// TwinCAT 3 PLC project _1_00
// ProgramVersion: 3.1.4023.0
// libraries:
//   Tc2_Standard, * (Beckhoff Automation GmbH)
//   Tc2_System, * (Beckhoff Automation GmbH)
//   Tc3_Module, * (Beckhoff Automation GmbH)
// project tree:
//   01_SubModule/01_Unit/ E_Unit.TcDUT, ST_Unit.TcDUT
//   01_SubModule/02_Station/ FB_Station.TcPOU
//   02_Module/ FB_Arm.TcPOU, FB_Barn.TcPOU, FB_Breeder.TcPOU, FB_Incubator.TcPOU, FB_Market.TcPOU
//   03_Game/ FB_Game.TcPOU
//   04_Main/ MAIN.TcPOU
//   / PlcTask.TcTTO
// real-time tasks:
//   TASK PlcTask: cycle T#10ms, priority 20, ADS port 350

CONFIGURATION _1_00
    RESOURCE PLC ON TwinCAT3
        TASK PlcTask(INTERVAL := T#10ms, PRIORITY := 20);
        PROGRAM MAIN WITH PlcTask : MAIN;
    END_RESOURCE
END_CONFIGURATION

// ---- 01_SubModule/01_Unit/E_Unit.TcDUT
{attribute 'qualified_only'}
{attribute 'strict'}
TYPE E_Unit :
(
	Invalid := -1,
	Egg		:= 0,
	Chicken	:= 1
):= Invalid;
END_TYPE

// ---- 01_SubModule/01_Unit/ST_Unit.TcDUT
TYPE ST_Unit :
STRUCT
	eType		: E_Unit;
	iHitPoint	: INT;
	iProgress	: INT;
END_STRUCT
END_TYPE

// ---- 04_Main/MAIN.TcPOU
PROGRAM MAIN
VAR
	(**)
	fbGame			: FB_Game;
	(*Button*)
	btStart			: BOOL;
	btPause			: BOOL;
	(*State*)
	GameRunning			: BOOL;
END_VAR

IF btStart THEN
	btStart := NOT btStart;
	GameRunning := TRUE;
END_IF

IF btPause THEN
	btPause := NOT btPause;
	GameRunning := FALSE;
END_IF

IF GameRunning THEN
	fbGame();
END_IF

END_PROGRAM

// ---- 03_Game/FB_Game.TcPOU
FUNCTION_BLOCK FB_Game
VAR
(*===========================================================================================================================*)
	(*Buttons*)
		(*Transfer*)
	btBarnToBreeder			: BOOL;
	btBarnToIncubator		: BOOL;
	btSellEgg				: BOOL;
	btSellChicken			: BOOL;
	btBreederToBarn			: BOOL;
	btPurchaseEgg			: BOOL;
	btPurchaseChicken		: BOOL;
		(*Upgrades*)
	btUpgradeArm			: BOOL;
	btUpgradeBarn			: BOOL;
	btUpgradeBreeder		: BOOL;
	btUpgradeIncubator		: BOOL;
	btUpgradeMarket			: BOOL;
	(*/Buttons*)
(*===========================================================================================================================*)
	(*Instance*)
		(*Stations*)
	fbBarn					: FB_Barn;
	fbBreeder				: FB_Breeder;
	fbIncubator				: FB_Incubator;
	fbMarket				: FB_Market;
		(*Arms*)
	fbArmArr				: ARRAY [1..5] OF FB_Arm;
	iCurArmLevel			: INT;
	iMaxArmLevel			: INT;
		(*Status*)
	iDay					: INT;
	iHour					: INT;
	iCurrency				: INT;
	iCost					: INT;
	iBarnUnit				: INT;
	iBreederUnit			: INT;
	iIncubatorUnit			: INT;
	iMarketUnit				: INT;
		(*Game Setting*)
	MaxStationLevel			: INT	:= 5;
	BarnLocation			: REAL	:= 10;
	BreederLocation			: REAL	:= 50;
	IncubatorLocation		: REAL	:= 90;
	MarketLocation			: REAL	:= 130;
	InitArmX				: REAL	:= 0;
	InitArmY				: REAL	:= 0;
	
		(*Timer*)
	fbTon60FPS				: TON;
	fbTon30FPS				: TON;
	fbTon1S					: TON;
	(*/Instance*)
END_VAR

Initialize(MaxStationLevel, BarnLocation, BreederLocation, IncubatorLocation, MarketLocation, 100);

fbTon30FPS(IN:= TRUE, PT:= T#33MS);
IF fbTon30FPS.Q THEN
	fbTon30FPS(IN:= FALSE);
	
	fbBarn.SortDescending();
	fbBreeder.SortAscending();
	fbIncubator.SortAscending();
	
	ButtonsTransfer();
	ArmRun();
	
	iBarnUnit := fbBarn.TotalUnit;
	iBreederUnit := fbBreeder.TotalUnit;
	iIncubatorUnit := fbIncubator.TotalUnit;
	iMarketUnit := fbMarket.TotalUnit;
	
END_IF

fbTon1S(IN:= TRUE, PT:= T#1S);
IF fbTon1S.Q THEN
	fbTon1S(IN:= FALSE);
	
	fbBarn.Run();
	fbBarn.HpRecover();
	
	fbBreeder.Run();
	fbBreeder.HpDeduct();
	
	fbIncubator.Run();
	
	fbMarket.Run();
	
	fbBarn.AutoImport(fbBreeder.Breeding(), fbIncubator.Hatching());
	iCurrency := iCurrency + fbMarket.Marketing();
	
	iHour := iHour + 1;
END_IF

IF iHour > 23 THEN
	iHour := 0;
	iDay := iDay + 1;
	iCurrency := iCurrency - iCost;
	IF iCurrency >= 0 THEN
		iCost := iCost + iDay*10;
	ELSE
		// Lose
	END_IF
	
END_IF

IF iDay > 30 THEN
	// Win
END_IF

METHOD ArmRun : PVOID
VAR
	iIndex			: INT;
END_VAR
fbArmArr[1].Run();
fbArmArr[2].Run();
fbArmArr[3].Run();
fbArmArr[4].Run();
fbArmArr[5].Run();

FOR iIndex := 1 TO iCurArmLevel BY 1 DO
	IF fbArmArr[iIndex].Load THEN
		IF
			fbArmArr[iIndex].CurX = fbBarn.Location THEN
			IF
				fbArmArr[iIndex].UnitType = 0 THEN
				fbArmArr[iIndex].CurUnit := fbBarn.UnitExport(0);
				fbArmArr[iIndex].Load := FALSE;
			ELSIF
				fbArmArr[iIndex].UnitType = 1 THEN
				fbArmArr[iIndex].CurUnit := fbBarn.UnitExport(1);
				fbArmArr[iIndex].Load := FALSE;
			END_IF
		ELSIF
			fbArmArr[iIndex].CurX = fbBreeder.Location THEN
			IF
				fbArmArr[iIndex].UnitType = 1 THEN
				fbArmArr[iIndex].CurUnit := fbBreeder.UnitExport(1);
				fbArmArr[iIndex].Load := FALSE;
			END_IF
		END_IF
	END_IF
END_FOR

FOR iIndex := 1 TO iCurArmLevel BY 1 DO
	IF fbArmArr[iIndex].Unload THEN
		IF
			fbArmArr[iIndex].CurX = fbBarn.Location THEN
			fbBarn.UnitImport(fbArmArr[iIndex].CurUnit);
			fbArmArr[iIndex].Unload := FALSE;
		ELSIF
			fbArmArr[iIndex].CurX = fbBreeder.Location THEN
			fbBreeder.UnitImport(fbArmArr[iIndex].CurUnit);
			fbArmArr[iIndex].Unload := FALSE;
		ELSIF
			fbArmArr[iIndex].CurX = fbIncubator.Location THEN
			fbIncubator.UnitImport(fbArmArr[iIndex].CurUnit);
			fbArmArr[iIndex].Unload := FALSE;
		ELSIF
			fbArmArr[iIndex].CurX = fbMarket.Location THEN
			fbMarket.UnitImport(fbArmArr[iIndex].CurUnit);
			fbArmArr[iIndex].Unload := FALSE;
		END_IF
	END_IF
END_FOR
END_METHOD

METHOD ButtonsTransfer : PVOID
VAR
	stTempUnit			: ST_Unit;
END_VAR
IF btBarnToBreeder THEN
	btBarnToBreeder := NOT btBarnToBreeder;
	
	IF NOT fbBreeder.IsFull AND fbBarn.HasChicken THEN
		TransferUnit(fbBarn.Location, fbBreeder.Location, 1);
	END_IF
END_IF

IF btBarnToIncubator THEN
	btBarnToIncubator := NOT btBarnToIncubator;
	
	IF NOT fbIncubator.IsFull AND fbBarn.HasEgg  THEN
		TransferUnit(fbBarn.Location, fbIncubator.Location, 0);
	END_IF
END_IF

IF btSellEgg THEN
	btSellEgg := NOT btSellEgg;
	
	IF NOT fbMarket.IsFull AND fbBarn.HasEgg THEN
		TransferUnit(fbBarn.Location, fbMarket.Location, 0);
	END_IF	
END_IF

IF btSellChicken THEN
	btSellChicken := NOT btSellChicken;
	
	IF NOT fbMarket.IsFull AND fbBarn.HasChicken THEN
		TransferUnit(fbBarn.Location, fbMarket.Location, 1);
	END_IF	
END_IF

IF btBreederToBarn THEN
	btBreederToBarn := NOT btBreederToBarn;
	
	IF NOT fbBarn.IsFull AND fbBreeder.HasChicken THEN
		TransferUnit(fbBreeder.Location, fbBarn.Location, 1);
	END_IF
END_IF

IF btPurchaseEgg THEN
	btPurchaseEgg := NOT btPurchaseEgg;
	
	IF NOT fbBarn.IsFull AND iCurrency > 20 THEN
		iCurrency := iCurrency - 20;
		
		stTempUnit.eType := 0;
		stTempUnit.iHitPoint := 30;
		stTempUnit.iProgress := 0;
		fbBarn.UnitImport(stTempUnit);
	END_IF
END_IF

IF btPurchaseChicken THEN
	btPurchaseChicken := NOT btPurchaseChicken;
	
	IF  NOT fbBarn.IsFull AND iCurrency > 12 THEN
		iCurrency := iCurrency - 12;
		
		stTempUnit.eType := 1;
		stTempUnit.iHitPoint := 30;
		stTempUnit.iProgress := 0;
		fbBarn.UnitImport(stTempUnit);
	END_IF
END_IF
END_METHOD

METHOD ButtonsUpgrade : PVOID
VAR_INPUT
END_VAR
IF btUpgradeArm THEN
	btUpgradeArm := NOT btUpgradeArm;
	
	IF iCurrency > (iCurArmLevel*30) THEN
		iCurrency := iCurrency - (iCurArmLevel*30);
		UpgradeArm(iCurArmLevel, InitArmX, InitArmY);
	END_IF
END_IF

IF btUpgradeBarn THEN
	btUpgradeBarn := NOT btUpgradeBarn;
	
	IF iCurrency > (fbBarn.Level*30) THEN
		iCurrency := iCurrency - (fbBarn.Level*30);
		fbBarn.Upgrade();
	END_IF
END_IF

IF btUpgradeBreeder THEN
	btUpgradeBreeder := NOT btUpgradeBreeder;
	
	IF iCurrency > (fbBreeder.Level*30) THEN
		iCurrency := iCurrency - (fbBreeder.Level*30);
		fbBreeder.Upgrade();
	END_IF
END_IF

IF btUpgradeIncubator THEN
	btUpgradeIncubator := NOT btUpgradeIncubator;
	
	IF iCurrency > (fbIncubator.Level*30) THEN
		iCurrency := iCurrency - (fbIncubator.Level*30);
		fbIncubator.Upgrade();
	END_IF
END_IF

IF btUpgradeMarket THEN
	btUpgradeMarket := NOT btUpgradeMarket;
	
	IF iCurrency > (fbMarket.Level*30) THEN
		iCurrency := iCurrency - (fbMarket.Level*30);
		fbMarket.Upgrade();
	END_IF
END_IF
END_METHOD

METHOD Initialize : PVOID
VAR_INPUT
	MaxLevel					: INT;
	BarnLocation				: REAL;
	BreederLocation				: REAL;
	IncubatorLocation			: REAL;
	MarketLocation				: REAL;
	Currency					: INT;
END_VAR
IF iDay = 0 THEN
	iDay := 1;
	
	fbBarn.Set(MaxLevel, BarnLocation);
	fbBreeder.Set(MaxLevel, BreederLocation);
	fbIncubator.Set(MaxLevel, IncubatorLocation);
	fbMarket.Set(MaxLevel, MarketLocation);
	UpgradeArm(iCurArmLevel, InitArmX, InitArmY);
	
	iCurrency := Currency;
	iCost := 10;
END_IF
END_METHOD

METHOD TransferUnit : PVOID
VAR_INPUT
	ImportLocation			: REAL;
	ExportLocation			: REAL;
	UnitType				: INT;	//0: Egg, 1: Chicken
END_VAR
VAR
	iIndex					: INT;
END_VAR
FOR iIndex := 1 TO iCurArmLevel BY 1 DO
	IF fbArmArr[iIndex].Activated AND NOT fbArmArr[iIndex].Busy THEN
		fbArmArr[iIndex].Assign(ImportLocation, ExportLocation, UnitType);
		RETURN;
	END_IF
END_FOR
END_METHOD

METHOD UpgradeArm : PVOID
VAR_INPUT
	CurrentArmIndex		: INT;
	InitX				: REAL;
	InitY				: REAL;
END_VAR
CurrentArmIndex := CurrentArmIndex + 1;
fbArmArr[CurrentArmIndex].Activated := TRUE;
fbArmArr[CurrentArmIndex].CurX := InitX;
fbArmArr[CurrentArmIndex].CurX := InitY;
iCurArmLevel := CurrentArmIndex;
END_METHOD

END_FUNCTION_BLOCK

// ---- 02_Module/FB_Barn.TcPOU
FUNCTION_BLOCK FB_Barn EXTENDS FB_Station
VAR
END_VAR

METHOD AutoImport : PVOID
VAR_INPUT
	Egg			: INT;
	Chicken		: INT;
END_VAR
VAR
	stTempEgg			: ST_Unit;
	iTempEgg			: INT;
	stTempChicken		: ST_Unit;
	iTempChicken		: INT;
END_VAR
FOR iTempEgg := 1 TO Egg BY 1 DO
	stTempEgg.eType := 0;
	stTempEgg.iHitPoint := 30;
	stTempEgg.iProgress := 0;
	UnitImport(stTempEgg);
END_FOR

FOR iTempChicken := 1 TO Chicken BY 1 DO
	stTempChicken.eType := 1;
	stTempChicken.iHitPoint := 30;
	stTempChicken.iProgress := 0;
	UnitImport(stTempChicken);
END_FOR
END_METHOD

METHOD Run : BOOL
VAR_INPUT
END_VAR
iMaxUnit := iCurLevel * 20;
END_METHOD

END_FUNCTION_BLOCK

// ---- 01_SubModule/02_Station/FB_Station.TcPOU
FUNCTION_BLOCK FB_Station
VAR
	stUnitArr			: ARRAY [1..100] OF ST_Unit;
	iMaxUnit			: INT;
	iLastIndex			: INT;
	
	iMaxLevel			: INT;
	iCurLevel			: INT := 1;
	
	rLocation			: REAL;
END_VAR

PROPERTY HasChicken : BOOL
GET
VAR
	iIndex			: INT;
END_VAR
HasChicken := FALSE;
IF iLastIndex > 0 THEN
	FOR iIndex := 1 TO iLastIndex BY 1 DO
		IF stUnitArr[iIndex].eType = 1 THEN
			HasChicken := NOT HasChicken;
			RETURN;
		END_IF
	END_FOR
END_IF
END_GET
END_PROPERTY

PROPERTY HasEgg : BOOL
GET
VAR
	iIndex			: INT;
END_VAR
HasEgg := FALSE;
IF iLastIndex > 0 THEN
	FOR iIndex := 1 TO iLastIndex BY 1 DO
		IF stUnitArr[iIndex].eType = 0 THEN
			HasEgg := NOT HasEgg;
			RETURN;
		END_IF
	END_FOR
END_IF
END_GET
END_PROPERTY

METHOD HpDeduct : PVOID
VAR
	iTempIndex			: INT;
END_VAR
IF iLastIndex < 1 THEN
	RETURN;
END_IF

FOR iTempIndex := 1 TO iLastIndex BY 1 DO
	stUnitArr[iTempIndex].iHitPoint := stUnitArr[iTempIndex].iHitPoint - 1;
	IF stUnitArr[iTempIndex].iHitPoint = 0 THEN
		RemoveUnit(iTempIndex);
	END_IF
END_FOR
END_METHOD

METHOD HpRecover : PVOID
VAR
	iTempIndex			: INT;
END_VAR
IF iLastIndex < 1 THEN
	RETURN;
END_IF

FOR iTempIndex := 1 TO iLastIndex BY 1 DO
	IF stUnitArr[iTempIndex].iHitPoint < 30 THEN
		stUnitArr[iTempIndex].iHitPoint := stUnitArr[iTempIndex].iHitPoint + 1;
	END_IF
END_FOR
END_METHOD

PROPERTY IsFull : BOOL
GET
IsFull := TRUE;
IF iLastIndex < iMaxUnit THEN
	IsFull := NOT IsFull;
END_IF
END_GET
END_PROPERTY

PROPERTY Level : INT
GET
Level := iCurLevel;
END_GET
END_PROPERTY

PROPERTY Location : REAL
GET
Location := rLocation;
END_GET
END_PROPERTY

METHOD RemoveUnit : PVOID
VAR_INPUT
	iIndex			: INT;
END_VAR
stUnitArr[iIndex] := stUnitArr[iLastIndex];
stUnitArr[iLastIndex].eType := -1;
stUnitArr[iLastIndex].iHitPoint := 0;
stUnitArr[iLastIndex].iProgress := 0;
iLastIndex := iLastIndex - 1;
END_METHOD

METHOD Run : BOOL
VAR_INPUT
END_VAR
iMaxUnit := iCurLevel * 10;
END_METHOD

METHOD Set : PVOID
VAR_INPUT
	MaxLevel			: INT;
	Location			: REAL;
END_VAR
iMaxLevel := MaxLevel;
rLocation := Location;
iCurLevel := 1;
END_METHOD

METHOD SortAscending : PVOID
VAR
	iCurIndex			: INT;
	stTempUnit			: ST_Unit;
	iTempIndex			: INT;
END_VAR
IF iLastIndex < 2 THEN
	RETURN;
END_IF

FOR iTempIndex := 1 TO iLastIndex BY 1 DO
	FOR iCurIndex := 1 TO iLastIndex BY 1 DO
		IF stUnitArr[iCurIndex].iHitPoint > stUnitArr[iTempIndex].iHitPoint THEN
			stTempUnit := stUnitArr[iCurIndex];
			stUnitArr[iCurIndex] := stUnitArr[iTempIndex];
			stUnitArr[iTempIndex] := stTempUnit;
		END_IF
	END_FOR
END_FOR
END_METHOD

METHOD SortDescending : PVOID
VAR
	iCurIndex			: INT;
	stTempUnit			: ST_Unit;
	iTempIndex			: INT;
END_VAR
IF iLastIndex < 2 THEN
	RETURN;
END_IF

FOR iTempIndex := 1 TO iLastIndex BY 1 DO
	FOR iCurIndex := 1 TO iLastIndex BY 1 DO
		IF stUnitArr[iCurIndex].iHitPoint < stUnitArr[iTempIndex].iHitPoint THEN
			stTempUnit := stUnitArr[iCurIndex];
			stUnitArr[iCurIndex] := stUnitArr[iTempIndex];
			stUnitArr[iTempIndex] := stTempUnit;
		END_IF
	END_FOR
END_FOR
END_METHOD

PROPERTY TotalUnit : INT
GET
TotalUnit := iLastIndex;
END_GET
END_PROPERTY

METHOD UnitExport : ST_Unit
VAR_INPUT
	UnitType			: INT; // 0: Egg, 1: Chicken
END_VAR
VAR
	iTempIndex			: INT;
END_VAR
IF iLastIndex < 1 THEN
	RETURN;
END_IF

CASE UnitType OF
	0: 
		FOR iTempIndex := 1 TO iLastIndex BY 1 DO
			IF stUnitArr[iTempIndex].eType = UnitType THEN
				stUnitArr[iTempIndex].iProgress := 0;
				UnitExport := stUnitArr[iTempIndex];
				stUnitArr[iTempIndex] := stUnitArr[iLastIndex];
				stUnitArr[iLastIndex].eType := -1;
				stUnitArr[iLastIndex].iHitPoint := 0;
				iLastIndex := iLastIndex - 1;
				RETURN;
			END_IF
		END_FOR
		
	1:
		FOR iTempIndex := 1 TO iLastIndex BY 1 DO
			IF stUnitArr[iTempIndex].eType = UnitType THEN
				stUnitArr[iTempIndex].iProgress := 0;
				UnitExport := stUnitArr[iTempIndex];
				stUnitArr[iTempIndex] := stUnitArr[iLastIndex];
				stUnitArr[iLastIndex].eType := -1;
				stUnitArr[iLastIndex].iHitPoint := 0;
				iLastIndex := iLastIndex - 1;
				RETURN;
			END_IF
		END_FOR
END_CASE
END_METHOD

METHOD UnitImport : PVOID
VAR_INPUT
	Unit			: ST_Unit;
END_VAR
IF Unit.eType <> -1 THEN
	IF iLastIndex < iMaxUnit THEN
		iLastIndex := iLastIndex + 1;
		stUnitArr[iLastIndex] := Unit;
	END_IF
END_IF
END_METHOD

METHOD Upgrade : PVOID
IF iCurLevel < iMaxLevel THEN
	iCurLevel := iCurLevel + 1;
END_IF
END_METHOD

END_FUNCTION_BLOCK

// ---- 02_Module/FB_Breeder.TcPOU
FUNCTION_BLOCK FB_Breeder EXTENDS FB_Station
VAR
	iBreedableArr			: ARRAY [1..50] OF INT;
	iLastBreedIndex			: INT;
END_VAR

METHOD Breeding : INT
VAR
	stTempUnit				: ST_Unit;
	iTempIndex				: INT;
	iBreedIndex				: INT;
	iBreedCounter			: INT;
END_VAR
Breeding := 0;
IF iLastIndex > 1 THEN
	FOR iTempIndex := 1 TO iLastIndex BY 1 DO
		stTempUnit := stUnitArr[iTempIndex];
		IF stTempUnit.iProgress < 6 THEN
			stTempUnit.iProgress := stTempUnit.iProgress + 1;
			stUnitArr[iTempIndex] := stTempUnit;
		ELSE
			iBreedIndex := iBreedIndex + 1;
			iBreedableArr[iBreedIndex] := iTempIndex;
			iLastBreedIndex := iBreedIndex;
		END_IF
	END_FOR
END_IF

IF iLastBreedIndex > 1 THEN
	FOR iBreedIndex := 1 TO iLastBreedIndex BY 1 DO
		stTempUnit := stUnitArr[iBreedableArr[iBreedIndex]];
		stTempUnit.iProgress := 0;
		stUnitArr[iBreedableArr[iBreedIndex]] := stTempUnit;
		iBreedCounter := iBreedCounter + 1;
	END_FOR
	iLastBreedIndex := 0;
	Breeding := iBreedCounter / 2;
END_IF
END_METHOD

END_FUNCTION_BLOCK

// ---- 02_Module/FB_Incubator.TcPOU
FUNCTION_BLOCK FB_Incubator EXTENDS FB_Station
VAR
END_VAR

METHOD Hatching : INT
VAR
	stTempUnit				: ST_Unit;
	iTempIndex				: INT;
	iHatchCounter			: INT;
END_VAR
Hatching := 0;
IF iLastIndex > 0 THEN
	FOR iTempIndex := 1 TO iLastIndex BY 1 DO
		stTempUnit := stUnitArr[iTempIndex];
		IF stTempUnit.iProgress < 6 THEN
			stTempUnit.iProgress := stTempUnit.iProgress + 1;
			stUnitArr[iTempIndex] := stTempUnit;
		ELSE
			RemoveUnit(iTempIndex);
			iHatchCounter := iHatchCounter + 1;
		END_IF
	END_FOR
END_IF
Hatching := iHatchCounter;
END_METHOD

END_FUNCTION_BLOCK

// ---- 02_Module/FB_Market.TcPOU
FUNCTION_BLOCK FB_Market EXTENDS FB_Station
VAR
END_VAR

METHOD Marketing : INT
VAR
	stTempUnit				: ST_Unit;
	iTempIndex				: INT;
	iSold					: INT;
END_VAR
Marketing := 0;
IF iLastIndex > 0 THEN
	FOR iTempIndex := 1 TO iLastIndex BY 1 DO
		stTempUnit := stUnitArr[iTempIndex];
		IF stTempUnit.iProgress < 6 THEN
			stTempUnit.iProgress := stTempUnit.iProgress + 1;
			stUnitArr[iTempIndex] := stTempUnit;
		ELSE
			IF stTempUnit.eType = 0 THEN
				Marketing := Marketing + 8;
			ELSIF 
				stTempUnit.eType = 1 THEN
				Marketing := Marketing + 15;
			END_IF
			RemoveUnit(iTempIndex);
		END_IF
	END_FOR
END_IF
END_METHOD

END_FUNCTION_BLOCK

// ---- 02_Module/FB_Arm.TcPOU
FUNCTION_BLOCK FB_Arm
VAR
	bActivated			: BOOL;
	bBusy				: BOOL;
	bRunning			: BOOL;
	bLoad				: BOOL;
	bUnload				: BOOL;
	
	rCurX				: REAL;
	rCurY				: REAL;
	
	rImportX			: REAL;
	rExportX			: REAL;
	rLoadingY			: REAL	:= 0;
	
	rIdleX				: REAL	:= 0;
	rIdleY				: REAL	:= 10;
	
	stUnit				: ST_Unit;
	
	iType				: INT;
	iCase				: INT;
END_VAR

PROPERTY Activated : BOOL
GET
Activated := bActivated;
END_GET
SET
bActivated := Activated;
END_SET
END_PROPERTY

METHOD Assign : PVOID
VAR_INPUT
	ImportLocation			: REAL;
	ExportLocation			: REAL;
	UnitType				: INT;
END_VAR
IF NOT bBusy AND bActivated THEN
	bBusy := TRUE;
	rImportX := ImportLocation;
	rExportX := ExportLocation;
	iType := UnitType;
END_IF
END_METHOD

PROPERTY Busy : BOOL
GET
Busy := bBusy;
END_GET
END_PROPERTY

PROPERTY CurUnit : ST_Unit
GET
CurUnit := stUnit;
stUnit.eType := -1;
END_GET
SET
IF CurUnit.eType <> -1 THEN
	stUnit := CurUnit;
END_IF
END_SET
END_PROPERTY

PROPERTY CurX : REAL
GET
CurX := rCurX;
END_GET
SET
rCurX := CurX;
END_SET
END_PROPERTY

PROPERTY CurY : REAL
GET
CurY := rCurY;
END_GET
SET
rCurY := CurY;
END_SET
END_PROPERTY

PROPERTY Load : BOOL
GET
Load := bLoad;
END_GET
SET
bLoad := Load;
END_SET
END_PROPERTY

METHOD Run : PVOID
VAR_INPUT
END_VAR
IF NOT bBusy THEN
	iCase := 0;
END_IF
IF bBusy AND NOT bRunning THEN
	bRunning := TRUE;
	iCase := 1;
END_IF

CASE iCase OF
	0:	(*Idle*)
		IF rCurY < rIdleY THEN
			rCurY := rCurY + 1;
		ELSIF
			rCurY > rIdleY THEN
			rCurY := rCurY - 1;
		ELSE
			IF rCurX < rIdleX THEN
				rCurX := rCurX + 1;
			ELSIF 
				rCurX > rIdleX THEN
				rCurX := rCurX - 1;
			END_IF
		END_IF
		
	1:	(*Go Import Location*)
		IF rCurY < rIdleY THEN
			rCurY := rCurY + 1;
		ELSIF
			rCurY > rIdleY THEN
			rCurY := rCurY - 1;
		ELSE
			IF rCurX < rImportX THEN
				rCurX := rCurX + 1;
			ELSIF
				rCurX > rImportX THEN
				rCurX := rCurX - 1;
			ELSE
				iCase := 11;
			END_IF
		END_IF
		
	11:	(*Go to Loading Position*)
		IF rCurY < rLoadingY THEN
			rCurY := rCurY + 1;
		ELSIF 
			rCurY > rLoadingY THEN
			rCurY := rCurY - 1;
		ELSE
			bLoad := TRUE;
			iCase := 2;
		END_IF
	
	2:	(*Load*)
		IF NOT bLoad THEN
			iCase := 3;
		END_IF
		
	21:	(*Leave Loading Position*)
		IF rCurY < rIdleY THEN
			rCurY := rCurY + 1;
		ELSIF
			rCurY > rIdleY THEN
			rCurY := rCurY - 1;
		ELSE
			iCase := 3;
		END_IF
	
	3:	(*Go to Export Location*)
		IF rCurX < rExportX THEN
			rCurX := rCurX + 1;
		ELSIF
			rCurX > rExportX THEN
			rCurX := rCurX - 1;
		ELSE
			IF rCurY < rLoadingY THEN
				rCurY := rCurY + 1;
			ELSIF 
				rCurY > rLoadingY THEN
				rCurY := rCurY - 1;
			ELSE
				bUnload := TRUE;
				iCase := 4;
			END_IF
		END_IF
		
	4:	(*Unload*)
		IF NOT bUnload THEN
			iCase := 0;
			bBusy := FALSE;
			bRunning := FALSE;
		END_IF
	
END_CASE
END_METHOD

PROPERTY UnitType : INT
GET
UnitType := iType;
END_GET
END_PROPERTY

PROPERTY Unload : BOOL
GET
Unload := bUnload;
END_GET
SET
bUnload := Unload;
END_SET
END_PROPERTY

END_FUNCTION_BLOCK
